FUNCTION_BLOCK FB_INFRATEC_TRIGERS
VAR_INPUT
END_VAR
VAR_OUTPUT
END_VAR
VAR
END_VAR

END_FUNCTION_BLOCK

(* stored: Version 1.1.0.1, ProductVersion 3.1.4024.12
   POU FB_INFRATEC_TRIGERS: Id {08f7d1b0-9e2b-467f-b539-777e64e3b2e8}, SpecialFunc None *)
